Universal Robots PolyScope program: d_to_a.urp

Program d_to_a (installation=string_planes directory=/programs/string_crossings createdIn=5.17.3 lastSavedIn=5.17.3 robotSerialNumber=20245501435)
Calibrated DH parameters: a=[0.000154, -0.137004, -0.385524, -0.00002, 0.000092, 0]; d=[0.162441, 211.794786, -230.585024, 18.923638, 0.099786, 0.09951]; alpha=[1.569493, -0.001902, 0.003874, 1.570111, -1.570167, 0]; deltaTheta=[0, -1.242934, 1.056292, 0.186646, 0.000002, 0.000001]
InitVariablesNode
Robot Program (runOnlyOnce=true)
  bow_section := 1
  If bow_section≟-1
    MoveJ speed 60 deg/s, acceleration 80 deg/s^2 (useActiveTCP=true) feature=Base
      Waypoint Waypoint_3 (Relative): relativeFromPosition TCP in base x=316.068 y=723.618 z=117.805 mm, rx=-1.5349 ry=-2.2387 rz=1.1274 rad; joints [-128.458, -21.869, 50.821, -72.933, -81.954, -152.854] deg; TCP offset x=28.21 y=-96.107 z=-99.69 mm, rx=0 ry=0 rz=0 rad; TCP in base x=277.256 y=734.024 z=156.889 mm, rx=1.7389 ry=2.3104 rz=-1.1078 rad; joints [-126.649, -28.123, 54.728, -74.617, -91.964, -141.814] deg
  ElseIf bow_section≟0
    MoveJ speed 60 deg/s, acceleration 80 deg/s^2 (useActiveTCP=true) feature=Base
      Waypoint Waypoint_4 (Relative): relativeFromPosition TCP in base x=329.63 y=457.702 z=123.03 mm, rx=-1.5368 ry=-2.1747 rz=1.1049 rad; joints [-145.135, -44.399, 100.427, -98.676, -90.57, -164.149] deg; TCP in base x=327.082 y=542.85 z=231.412 mm, rx=1.6821 ry=2.3247 rz=-1.1115 rad; joints [-139.551, -50.206, 85.865, -84.66, -102.288, -153.001] deg
  Else 
    MoveJ speed 60 deg/s, acceleration 80 deg/s^2 (useActiveTCP=true) feature=Base
      Waypoint Waypoint_1 (Relative): relativeFromPosition TCP in base x=340.803 y=238.631 z=127.342 mm, rx=-1.5375 ry=-2.1223 rz=1.0863 rad; joints [-167.853, -53.469, 123.568, -113.681, -104.544, -179.465] deg; TCP in base x=374.961 y=359.138 z=303.027 mm, rx=1.6274 ry=2.3373 rz=-1.1146 rad; joints [-156.115, -66.367, 101.552, -88.732, -114.429, -168.117] deg
